FUNCTION_BLOCK SupplyAirControl
VAR_INPUT
	EN: BOOL;
END_VAR
VAR_OUTPUT
	ENO: BOOL;
	Recirculation: BOOL;
END_VAR
VAR
END_VAR

ENO := EN;

END_FUNCTION_BLOCK

(* stored: Version 1.1.0.1, ProductVersion 3.1.4024.3
   POU SupplyAirControl: Id {31324594-6c68-4323-994e-89f11b3364f4}, SpecialFunc None *)
